// TIA Portal project "IrrigatoreFB" (V16)

(* hardware
DEVICE "S7-1200 station_1"  S7-1200 Station
   slot 0: "Telaio di montaggio_0"  S7-1200 Rack  Rack  V1.0
   slot 1: "PLC_1"  CPU 1214C DC/DC/DC  6ES7 214-1AG40-0XB0  V4.1
*)

// ===== PLC "PLC_1"  CPU 1214C DC/DC/DC =====

VAR_GLOBAL   // PLC tag table "Tabella delle variabili standard"
   "UMIDITY_1" AT %I0.0 : Bool;
   "OPEN_1" AT %Q0.0 : Bool;
   "UMIDITY_2" AT %I0.1 : Bool;
   "UMIDITY_3" AT %I0.2 : Bool;
   "OPEN_2" AT %Q0.1 : Bool;
   "OPEN_3" AT %Q0.2 : Bool;
END_VAR

VAR_GLOBAL CONSTANT   // PLC tag table "Tabella delle variabili standard"
   "TEMPO_TRASCORSO_T_ON_1_Irrigatore1" : Time := T#3s;
   "TEMPO_TRASCORSO_T_ON_2_Irrigatore1" : Time := T#8s;
   "TEMPO_TRASCORSO_T_Pausa_Irrigatore1" : Time := T#10s;
   "TEMPO_TRASCORSO_T_ON_1_Irrigatore2" : Time := T#5s;
   "TEMPO_TRASCORSO_T_ON_2_Irrigatore2" : Time := T#10s;
   "TEMPO_TRASCORSO_T_Pausa_Irrigatore2" : Time := T#12s;
   "TEMPO_TRASCORSO_T_ON_1_Irrigatore3" : Time := T#7s;
   "TEMPO_TRASCORSO_T_ON_2_Irrigatore3" : Time := T#12s;
   "TEMPO_TRASCORSO_T_Pausa_Irrigatore3" : Time := T#14s;
END_VAR

DATA_BLOCK "Irrigatore_DB_1"   // DB1
{ S7_Optimized_Access := 'TRUE' }
VERSION : 0.1
// stored: InstanceOfName Irrigatore
"Irrigatore"
BEGIN
END_DATA_BLOCK

DATA_BLOCK "Irrigatore_DB_2"   // DB2
{ S7_Optimized_Access := 'TRUE' }
VERSION : 0.1
// stored: InstanceOfName Irrigatore
"Irrigatore"
BEGIN
END_DATA_BLOCK

DATA_BLOCK "Irrigatore_DB_3"   // DB3
{ S7_Optimized_Access := 'TRUE' }
VERSION : 0.1
// stored: InstanceOfName Irrigatore
"Irrigatore"
BEGIN
END_DATA_BLOCK

FUNCTION_BLOCK "Irrigatore"   // FB1, LAD
{ S7_Optimized_Access := 'TRUE' }
VERSION : 0.1
   VAR_INPUT
      UMIDITY : Bool;
      TEMPO_TRASCORSO_T_ON_1 : Time;
      TEMPO_TRASCORSO_T_ON_2 : Time;
      TEMPO_TRASCORSO_T_Pausa : Time;
   END_VAR
   VAR_OUTPUT
      OPEN : Bool;
   END_VAR
   VAR RETAIN
      HOME : Bool := true;
      ACTIVE_IRRIGATION : Bool;
      STOP_IRRIGATION : Bool;
      REACTIVE_IRRIGATION : Bool;
      IEC_Timer_0_Instance_1 : TON_TIME;
      IEC_Timer_0_Instance_2 : TON_TIME;
      IEC_Timer_0_Instance_3 : TON_TIME;
   END_VAR
BEGIN

REGION Network 1
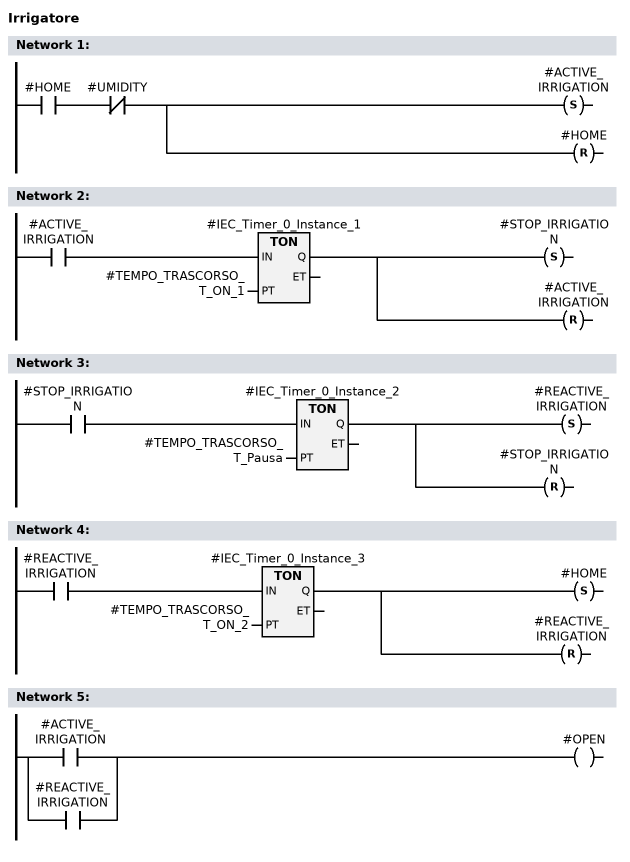
   RUNG wire#powerrail
      Contact( #HOME )
      I_Contact( #UMIDITY )
      wire#w1
      S_Coil( #ACTIVE_IRRIGATION )
   END_RUNG
   RUNG wire#w1
      R_Coil( #HOME )
   END_RUNG
   // the same network as SCL:
   IF #HOME AND NOT #UMIDITY THEN
       #ACTIVE_IRRIGATION := TRUE;
       #HOME := FALSE;
   END_IF;
END_REGION

REGION Network 2
   #IEC_Timer_0_Instance_1(IN := #ACTIVE_IRRIGATION, PT := #TEMPO_TRASCORSO_T_ON_1);   // TON
   IF #IEC_Timer_0_Instance_1.Q THEN
       #STOP_IRRIGATION := TRUE;
       #ACTIVE_IRRIGATION := FALSE;
   END_IF;
END_REGION

REGION Network 3
   #IEC_Timer_0_Instance_2(IN := #STOP_IRRIGATION, PT := #TEMPO_TRASCORSO_T_Pausa);   // TON
   IF #IEC_Timer_0_Instance_2.Q THEN
       #REACTIVE_IRRIGATION := TRUE;
       #STOP_IRRIGATION := FALSE;
   END_IF;
END_REGION

REGION Network 4
   #IEC_Timer_0_Instance_3(IN := #REACTIVE_IRRIGATION, PT := #TEMPO_TRASCORSO_T_ON_2);   // TON
   IF #IEC_Timer_0_Instance_3.Q THEN
       #HOME := TRUE;
       #REACTIVE_IRRIGATION := FALSE;
   END_IF;
END_REGION

REGION Network 5
   RUNG wire#powerrail
      Contact( #ACTIVE_IRRIGATION )
      wire#w1
      Coil( #OPEN )
   END_RUNG
   RUNG wire#powerrail
      Contact( #REACTIVE_IRRIGATION )
   END_RUNG wire#w1
   // the same network as SCL:
   #OPEN := #ACTIVE_IRRIGATION OR #REACTIVE_IRRIGATION;
END_REGION
END_FUNCTION_BLOCK

ORGANIZATION_BLOCK "Main"   // OB1, LAD, ProgramCycle
TITLE = "Main Program Sweep (Cycle)"
{ S7_Optimized_Access := 'TRUE' }
VERSION : 0.1
   VAR_INPUT
      Initial_Call : Bool;   // Initial call of this OB
      Remanence : Bool;   // =True, if remanent data are available
   END_VAR
BEGIN
END_ORGANIZATION_BLOCK

ORGANIZATION_BLOCK "Cyclic_Interrupt_50ms"   // OB30, LAD, CyclicInterrupt
{ S7_Optimized_Access := 'TRUE' }
VERSION : 0.1
   VAR_INPUT
      Initial_Call : Bool;   // Initial call of this OB
      Event_Count : Int;   // Events discarded
   END_VAR
BEGIN

REGION Network 1
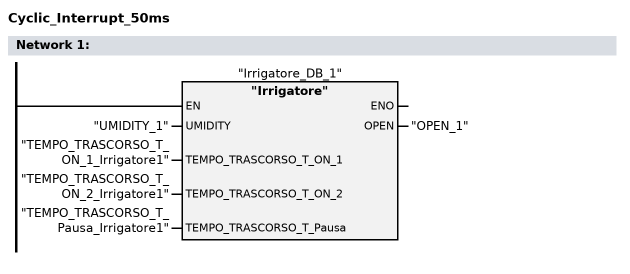
   RUNG wire#powerrail
      "Irrigatore_DB_1"(UMIDITY := "UMIDITY_1", TEMPO_TRASCORSO_T_ON_1 := "TEMPO_TRASCORSO_T_ON_1_Irrigatore1", TEMPO_TRASCORSO_T_ON_2 := "TEMPO_TRASCORSO_T_ON_2_Irrigatore1", TEMPO_TRASCORSO_T_Pausa := "TEMPO_TRASCORSO_T_Pausa_Irrigatore1", OPEN => "OPEN_1")
   END_RUNG
   // the same network as SCL:
   "Irrigatore_DB_1"(UMIDITY := "UMIDITY_1",   // "Irrigatore"
                     TEMPO_TRASCORSO_T_ON_1 := "TEMPO_TRASCORSO_T_ON_1_Irrigatore1",
                     TEMPO_TRASCORSO_T_ON_2 := "TEMPO_TRASCORSO_T_ON_2_Irrigatore1",
                     TEMPO_TRASCORSO_T_Pausa := "TEMPO_TRASCORSO_T_Pausa_Irrigatore1",
                     OPEN => "OPEN_1");
END_REGION
END_ORGANIZATION_BLOCK

ORGANIZATION_BLOCK "Cyclic_Interrupt_100ms"   // OB31, LAD, CyclicInterrupt
{ S7_Optimized_Access := 'TRUE' }
VERSION : 0.1
   VAR_INPUT
      Initial_Call : Bool;   // Initial call of this OB
      Event_Count : Int;   // Events discarded
   END_VAR
BEGIN

REGION Network 1
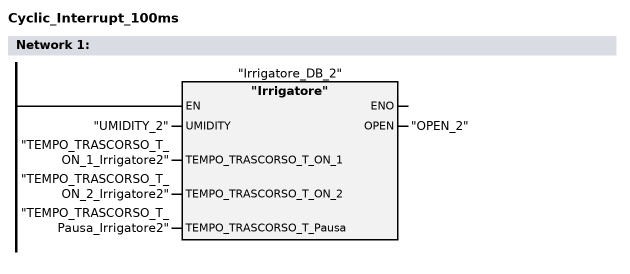
   RUNG wire#powerrail
      "Irrigatore_DB_2"(UMIDITY := "UMIDITY_2", TEMPO_TRASCORSO_T_ON_1 := "TEMPO_TRASCORSO_T_ON_1_Irrigatore2", TEMPO_TRASCORSO_T_ON_2 := "TEMPO_TRASCORSO_T_ON_2_Irrigatore2", TEMPO_TRASCORSO_T_Pausa := "TEMPO_TRASCORSO_T_Pausa_Irrigatore2", OPEN => "OPEN_2")
   END_RUNG
   // the same network as SCL:
   "Irrigatore_DB_2"(UMIDITY := "UMIDITY_2",   // "Irrigatore"
                     TEMPO_TRASCORSO_T_ON_1 := "TEMPO_TRASCORSO_T_ON_1_Irrigatore2",
                     TEMPO_TRASCORSO_T_ON_2 := "TEMPO_TRASCORSO_T_ON_2_Irrigatore2",
                     TEMPO_TRASCORSO_T_Pausa := "TEMPO_TRASCORSO_T_Pausa_Irrigatore2",
                     OPEN => "OPEN_2");
END_REGION
END_ORGANIZATION_BLOCK

ORGANIZATION_BLOCK "Cyclic_Interrupt_150ms"   // OB32, LAD, CyclicInterrupt
{ S7_Optimized_Access := 'TRUE' }
VERSION : 0.1
   VAR_INPUT
      Initial_Call : Bool;   // Initial call of this OB
      Event_Count : Int;   // Events discarded
   END_VAR
BEGIN

REGION Network 1
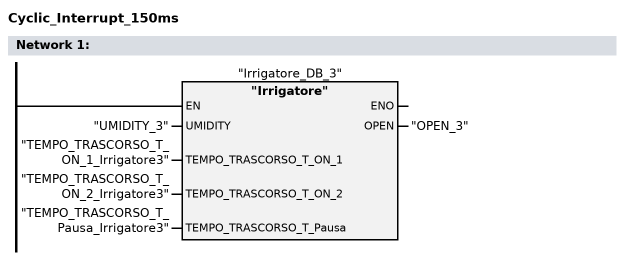
   RUNG wire#powerrail
      "Irrigatore_DB_3"(UMIDITY := "UMIDITY_3", TEMPO_TRASCORSO_T_ON_1 := "TEMPO_TRASCORSO_T_ON_1_Irrigatore3", TEMPO_TRASCORSO_T_ON_2 := "TEMPO_TRASCORSO_T_ON_2_Irrigatore3", TEMPO_TRASCORSO_T_Pausa := "TEMPO_TRASCORSO_T_Pausa_Irrigatore3", OPEN => "OPEN_3")
   END_RUNG
   // the same network as SCL:
   "Irrigatore_DB_3"(UMIDITY := "UMIDITY_3",   // "Irrigatore"
                     TEMPO_TRASCORSO_T_ON_1 := "TEMPO_TRASCORSO_T_ON_1_Irrigatore3",
                     TEMPO_TRASCORSO_T_ON_2 := "TEMPO_TRASCORSO_T_ON_2_Irrigatore3",
                     TEMPO_TRASCORSO_T_Pausa := "TEMPO_TRASCORSO_T_Pausa_Irrigatore3",
                     OPEN => "OPEN_3");
END_REGION
END_ORGANIZATION_BLOCK